(* PLC project Cell Example , CTH FIX1 1.0, author CTH SS2 *)
(* stored: companyURL www.chalmers.se, creationDateTime 2009-02-02T14:10:51, version 1.0, modificationDateTime 2009-02-12T12:58:33, organization SS2, language en-US *)

PROGRAM IL_Test
  VAR
    A : BOOL := false;
    B : BOOL := false;
    C : BOOL := false;
    G : BOOL := false;
    F : BOOL := false;
    H : BOOL := false;
    I : BOOL := false;
    J : BOOL := false;
    K : BOOL := false;
    M : BOOL := false;
    Q : BOOL := false;
    V1 : BOOL := false;
    V2 : BOOL := false;
    V3 : BOOL := false;
    V4 : BOOL := false;
  END_VAR

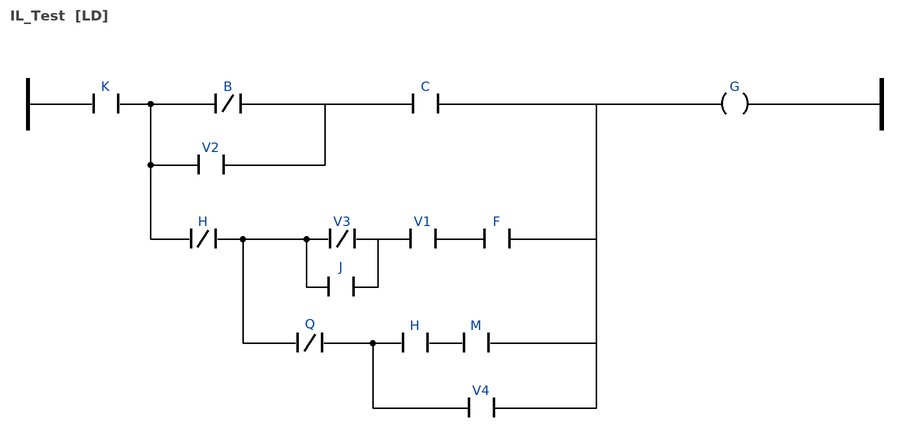
(* LD diagram, written out as Structured Text *)
G := K AND ((NOT B OR V2) AND C OR NOT H AND (NOT V3 OR J) AND V1 AND F OR NOT H AND NOT Q AND H AND M OR NOT H AND NOT Q AND V4);
END_PROGRAM
